SUBAPPLICATION Uebung_012e_AR (* Numeric Value Input PHYS und Speichern INI mit Subapp (AR Adapter) *)
  (* Standard: 61499-2; Description: Copyright (c) 2026 Meisterschulen am Ostbahnhof This program and the accompanying materials are made available under the terms of the Eclipse Public License 2.0 which is available at https://www.eclipse.org/legal/epl-2.0/ SPDX-License-Identifier: EPL-2.0 *)
  (* Version 1.0, 2026-04-24, Franz Höpfinger, Meisterschulen am Ostbahnhof, AR adapter variant of Uebung_012e *)
  PACKAGE Uebungen;
  IMPORT Uebungen::const::NVS::NVS_Keys::KEY_I1_STORE;
  IMPORT Uebungen::const::NVS::NVS_Keys::SECTION_I1_STORE;
  IMPORT Uebungen::const::UT::DefaultPool_Numeric::InputNumber_I1_N;
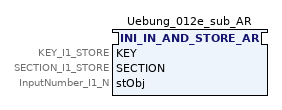
  SUBAPPS
    Uebung_012e_sub_AR : MyLib::sys::INI_IN_AND_STORE_AR(KEY := KEY_I1_STORE, SECTION := SECTION_I1_STORE, stObj := InputNumber_I1_N);
  END_SUBAPPS
END_SUBAPPLICATION
